(* CoDeSys 2.3.9.59 project: scope.pro *)
(* Libraries: STANDARD.LIB 5.6.98 11:03:02 *)

(* Task configuration *)
TASK Standard (PRIORITY := 0, INTERVAL := T#1ms);
	MAIN
END_TASK

(* Global variable list: TwinCAT_Configuration *)
(* Generated automatically by TwinCAT - (read only) *)
VAR_CONFIG
	MAIN.di_set_pos AT %QB0 : DINT;
END_VAR

(* POU MAIN, ST *)
PROGRAM MAIN
VAR
	(* nc *)
	fb_channel_set_pos	:fb_axis_simulator;

	di_set_pos			AT%Q*	:DINT;
	lr_set_pos					:LREAL;

	(* plc *)
	fb_channel_1			:fb_axis_simulator;
	fb_channel_2			:fb_axis_simulator;
	fb_channel_3			:fb_axis_simulator;
	fb_channel_4			:fb_axis_simulator;
	fb_channel_5			:fb_axis_simulator;
	fb_channel_6			:fb_axis_simulator;
	fb_channel_7			:fb_axis_simulator;
	fb_channel_8			:fb_axis_simulator;

	lr_channel_1			:LREAL;
	lr_channel_2			:LREAL;
	lr_channel_3			:LREAL;
	lr_channel_4			:LREAL;
	lr_channel_5			:LREAL;
	lr_channel_6			:LREAL;
	lr_channel_7			:LREAL;
	lr_channel_8			:LREAL;
END_VAR
(* nc *)
fb_channel_set_pos(
	l_t_impuls	:= t#1ms,
	i_i_range		:= 10000,
	i_lr_min		:= 0,
	i_lr_max		:= 1000000,
	io_lr_value	:= lr_set_pos);
di_set_pos := LREAL_TO_DINT(lr_set_pos);

(* plc *)
fb_channel_1(
	l_t_impuls	:= t#1ms,
	i_i_range		:= 2,
	i_lr_min		:= 0,
	i_lr_max		:= 100,
	io_lr_value	:= lr_channel_1);

fb_channel_2(
	l_t_impuls	:= t#1ms,
	i_i_range		:= 1,
	i_lr_min		:= 0,
	i_lr_max		:= 50,
	io_lr_value	:= lr_channel_2);

fb_channel_3(
	l_t_impuls	:= t#1ms,
	i_i_range		:= 8,
	i_lr_min		:= -400,
	i_lr_max		:= 0,
	io_lr_value	:= lr_channel_3);

fb_channel_4(
	l_t_impuls	:= t#1ms,
	i_i_range		:= 5,
	i_lr_min		:= 0,
	i_lr_max		:= 250,
	io_lr_value	:= lr_channel_4);

fb_channel_5(
	l_t_impuls	:= t#1ms,
	i_i_range		:= 5,
	i_lr_min		:= -250,
	i_lr_max		:= 0,
	io_lr_value	:= lr_channel_5);

fb_channel_6(
	l_t_impuls	:= t#1ms,
	i_i_range		:= 4,
	i_lr_min		:= 0,
	i_lr_max		:= 200,
	io_lr_value	:= lr_channel_6);

fb_channel_7(
	l_t_impuls	:= t#1ms,
	i_i_range		:= 10,
	i_lr_min		:= 0,
	i_lr_max		:= 500,
	io_lr_value	:= lr_channel_7);

fb_channel_8(
	l_t_impuls	:= t#1ms,
	i_i_range		:= 10,
	i_lr_min		:= -500,
	i_lr_max		:= 0,
	io_lr_value	:= lr_channel_8);
END_PROGRAM

(* POU fb_axis_simulator, ST *)
FUNCTION_BLOCK fb_axis_simulator

VAR_IN_OUT
	io_lr_value		:LREAL;
END_VAR

VAR_INPUT
	l_t_impuls		:TIME;
	i_i_range			:INT;
	i_lr_min			:LREAL;
	i_lr_max			:LREAL;
END_VAR

VAR
	l_ton_timer		:TON;
	l_b_impuls		:BOOL;
	l_b_direction		:BOOL;
END_VAR
l_ton_timer( PT := l_t_impuls );

IF l_ton_timer.Q THEN
	l_ton_timer.IN := FALSE;
ELSE
	l_ton_timer.IN := TRUE;
END_IF

IF io_lr_value > i_lr_max THEN
	l_b_direction := TRUE;
END_IF

IF io_lr_value < i_lr_min THEN
	l_b_direction := FALSE;
END_IF

IF  l_ton_timer.Q THEN
	IF l_b_direction THEN
		io_lr_value := io_lr_value - i_i_range;
	ELSE
		io_lr_value := io_lr_value + i_i_range;
	END_IF
END_IF
END_FUNCTION_BLOCK
